TYPE IOL_4IN :
STRUCT
	BYTE0	AT %I* 	: USINT;
    BYTE1	AT %I* 	: USINT;
    BYTE2	AT %I* 	: USINT;
    BYTE3	AT %I* 	: USINT;
END_STRUCT
END_TYPE

(* stored: Version 1.1.0.1
   DUT IOL_4IN: Id {016e1223-2d69-48e0-b2b0-3f7df97a0ec2} *)
